// TIA Portal project "Traffic Light Controller" (V16)

(* hardware
DEVICE "S7-1200 station_1"  S7-1200 Station
   slot 0: "Rack_0"  S7-1200 Rack  Rack  V1.0
   slot 1: "PLC_1"  CPU 1212C DC/DC/DC  6ES7 212-1AE40-0XB0  V4.4
DEVICE "HMI_1"  TP700 Comfort
   slot 0: "HMI_1"  TP700 Comfort  6AV2 124-0GC01-0AX0  16.0.0.0
   slot 1: "HMI_RT_1"  TP700 Comfort  6AV2 124-0GC01-0AX0  16.0.0.0
   slot 5: "HMI_1.IE_CP_1"  PROFINET Interface  16.0.0.0
      slot 1: "PROFINET Interface_1"  PROFINET Interface
         slot 1: "Port_1"  Port
         slot 2: "Port_2"  Port
   slot 7: "HMI_1.MPI/DP_CP_1"  MPI/DP Interface  16.0.0.0
*)

// ===== PLC "PLC_1"  CPU 1212C DC/DC/DC =====

VAR_GLOBAL   // PLC tag table "Tag table_1"
   "START" AT %M0.0 : Bool;
   "STOP" AT %M0.1 : Bool;
   "STARTED" AT %M0.2 : Bool;
   "STEP1_EAST_GREEN" AT %M0.3 : Bool;
   "STEP1_WEST_RED" AT %M0.4 : Bool;
   "STEP1_NORTH_RED" AT %M0.5 : Bool;
   "STEP1_EAST_YELLOW" AT %M0.6 : Bool;
   "STEP1_FINISHED" AT %M0.7 : Bool;
   "STEP2_WEST_GREEN" AT %M1.0 : Bool;
   "STEP2_EAST_RED" AT %M1.1 : Bool;
   "STEP2_NORTH_RED" AT %M1.2 : Bool;
   "STEP2_WEST_YELLOW" AT %M1.3 : Bool;
   "STEP2_FINISHED" AT %M1.4 : Bool;
   "STEP3_NORTH_GREEN" AT %M1.5 : Bool;
   "STEP3_EAST_RED" AT %M1.6 : Bool;
   "STEP3_WEST_RED" AT %M1.7 : Bool;
   "STEP3_NORTH_YELLOW" AT %M2.0 : Bool;
   "STEP3_FINISHED" AT %M2.1 : Bool;
   "EAST_GREEN" AT %M2.2 : Bool;
   "EAST_RED" AT %M2.4 : Bool;
   "NORTH_RED" AT %M2.5 : Bool;
   "NORTH_YELLOW" AT %M2.6 : Bool;
   "NORTH_GREEN" AT %M2.7 : Bool;
   "WEST_RED" AT %M3.0 : Bool;
   "WEST_GREEN" AT %M3.1 : Bool;
   "WEST_YELLOW" AT %M3.2 : Bool;
   "EAST_YELLOW" AT %M2.3 : Bool;
END_VAR

// folder: System blocks/Program resources

DATA_BLOCK "STEP1"   // DB1
{ S7_Optimized_Access := 'TRUE' }
AUTHOR : Simatic
FAMILY : IEC
NAME : IEC_TMR
VERSION : 1.0
// stored: InstanceOfName IEC_TIMER
"IEC_TIMER"
BEGIN
END_DATA_BLOCK

DATA_BLOCK "COUNTER_STEP"   // DB2
{ S7_Optimized_Access := 'TRUE' }
AUTHOR : Simatic
FAMILY : IEC
NAME : CNTR
VERSION : 1.0
// stored: InstanceOfName IEC_COUNTER
"IEC_COUNTER"
BEGIN
END_DATA_BLOCK

DATA_BLOCK "STEP2"   // DB3
{ S7_Optimized_Access := 'TRUE' }
AUTHOR : Simatic
FAMILY : IEC
NAME : IEC_TMR
VERSION : 1.0
// stored: InstanceOfName IEC_TIMER
"IEC_TIMER"
BEGIN
END_DATA_BLOCK

DATA_BLOCK "STEP3"   // DB4
{ S7_Optimized_Access := 'TRUE' }
AUTHOR : Simatic
FAMILY : IEC
NAME : IEC_TMR
VERSION : 1.0
// stored: InstanceOfName IEC_TIMER
"IEC_TIMER"
BEGIN
END_DATA_BLOCK

// folder: (top level)

ORGANIZATION_BLOCK "Main"   // OB1, LAD, ProgramCycle
TITLE = "Main Program Sweep (Cycle)"
{ S7_Optimized_Access := 'TRUE' }
VERSION : 0.1
   VAR_INPUT
      Initial_Call : Bool;   // Initial call of this OB
      Remanence : Bool;   // =True, if remanent data are available
   END_VAR
   VAR_TEMP   // added for the SCL form of the ladder/FBD networks
      _w1 : Bool;
      _w2 : Bool;
      _w3 : Bool;
   END_VAR
BEGIN

REGION Network 1
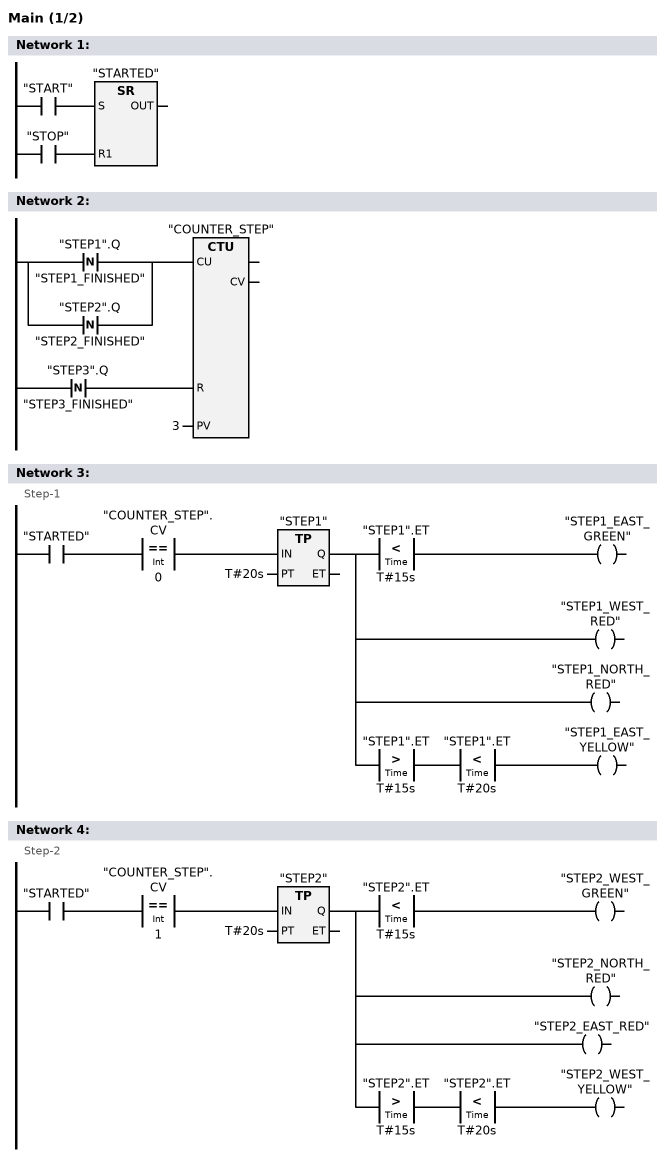
   RUNG wire#powerrail
      Contact( "START" )
      S_SR(operand := "STARTED", r1 := wire#w1)
   END_RUNG
   RUNG wire#powerrail
      Contact( "STOP" )
   END_RUNG wire#w1
   // the same network as SCL:
   IF "START" THEN
       "STARTED" := TRUE;   // SR flip-flop
   END_IF;
   IF "STOP" THEN "STARTED" := FALSE; END_IF;
END_REGION

REGION Network 2
   #_w1 := NOT "STEP1".Q AND "STEP1_FINISHED";   // falling edge of "STEP1".Q
   "STEP1_FINISHED" := "STEP1".Q;
   #_w2 := NOT "STEP2".Q AND "STEP2_FINISHED";   // falling edge of "STEP2".Q
   "STEP2_FINISHED" := "STEP2".Q;
   #_w3 := NOT "STEP3".Q AND "STEP3_FINISHED";   // falling edge of "STEP3".Q
   "STEP3_FINISHED" := "STEP3".Q;
   "COUNTER_STEP".CTU(CU := #_w1 OR #_w2, R := #_w3, PV := 3);
END_REGION

REGION Network 3
   // Step-1
   "STEP1".TP(IN := "STARTED" AND ("COUNTER_STEP".CV = 0), PT := T#20s);
   "STEP1_EAST_GREEN" := "STEP1".Q AND ("STEP1".ET < T#15s);
   "STEP1_WEST_RED" := "STEP1".Q;
   "STEP1_NORTH_RED" := "STEP1".Q;
   "STEP1_EAST_YELLOW" := "STEP1".Q AND ("STEP1".ET > T#15s) AND ("STEP1".ET < T#20s);
END_REGION

REGION Network 4
   // Step-2
   "STEP2".TP(IN := "STARTED" AND ("COUNTER_STEP".CV = 1), PT := T#20s);
   "STEP2_WEST_GREEN" := "STEP2".Q AND ("STEP2".ET < T#15s);
   "STEP2_NORTH_RED" := "STEP2".Q;
   "STEP2_EAST_RED" := "STEP2".Q;
   "STEP2_WEST_YELLOW" := "STEP2".Q AND ("STEP2".ET > T#15s) AND ("STEP2".ET < T#20s);
END_REGION

REGION Network 5
   // Step-3
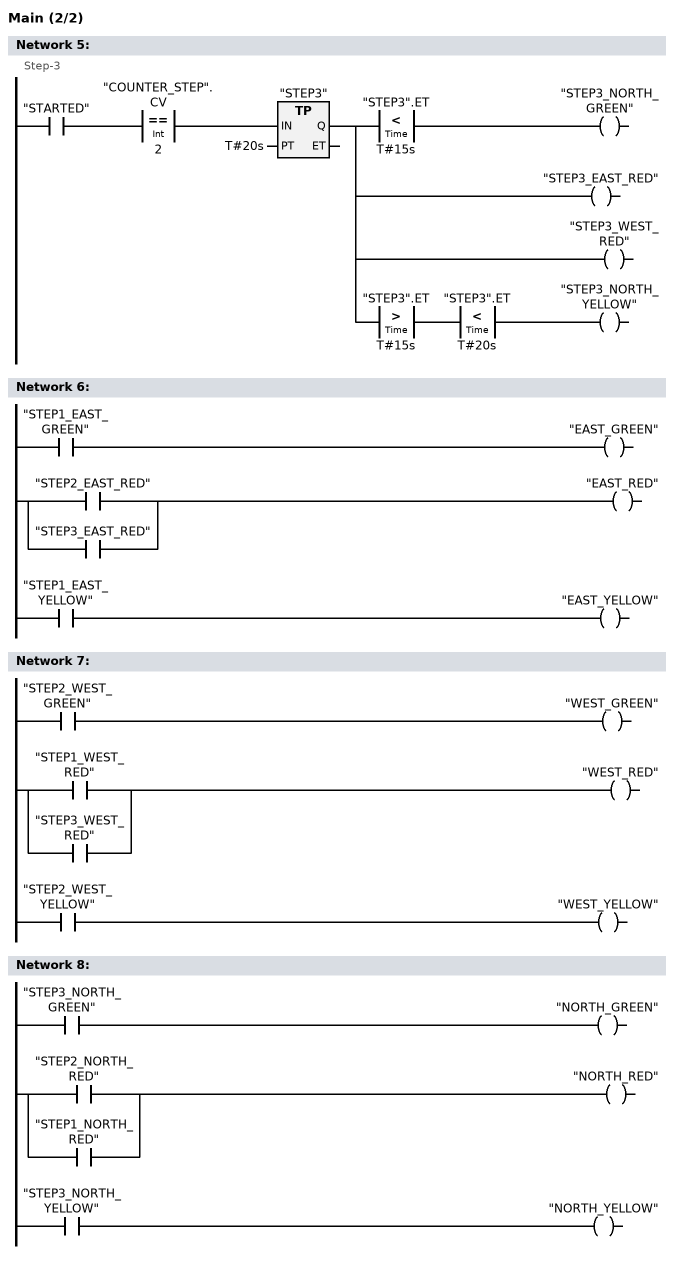
   "STEP3".TP(IN := "STARTED" AND ("COUNTER_STEP".CV = 2), PT := T#20s);
   "STEP3_NORTH_GREEN" := "STEP3".Q AND ("STEP3".ET < T#15s);
   "STEP3_EAST_RED" := "STEP3".Q;
   "STEP3_WEST_RED" := "STEP3".Q;
   "STEP3_NORTH_YELLOW" := "STEP3".Q AND ("STEP3".ET > T#15s) AND ("STEP3".ET < T#20s);
END_REGION

REGION Network 6
   RUNG wire#powerrail
      Contact( "STEP1_EAST_GREEN" )
      Coil( "EAST_GREEN" )
   END_RUNG
   RUNG wire#powerrail
      Contact( "STEP2_EAST_RED" )
      wire#w1
      Coil( "EAST_RED" )
   END_RUNG
   RUNG wire#powerrail
      Contact( "STEP3_EAST_RED" )
   END_RUNG wire#w1
   RUNG wire#powerrail
      Contact( "STEP1_EAST_YELLOW" )
      Coil( "EAST_YELLOW" )
   END_RUNG
   // the same network as SCL:
   "EAST_GREEN" := "STEP1_EAST_GREEN";
   "EAST_RED" := "STEP2_EAST_RED" OR "STEP3_EAST_RED";
   "EAST_YELLOW" := "STEP1_EAST_YELLOW";
END_REGION

REGION Network 7
   RUNG wire#powerrail
      Contact( "STEP2_WEST_GREEN" )
      Coil( "WEST_GREEN" )
   END_RUNG
   RUNG wire#powerrail
      Contact( "STEP1_WEST_RED" )
      wire#w1
      Coil( "WEST_RED" )
   END_RUNG
   RUNG wire#powerrail
      Contact( "STEP3_WEST_RED" )
   END_RUNG wire#w1
   RUNG wire#powerrail
      Contact( "STEP2_WEST_YELLOW" )
      Coil( "WEST_YELLOW" )
   END_RUNG
   // the same network as SCL:
   "WEST_GREEN" := "STEP2_WEST_GREEN";
   "WEST_RED" := "STEP1_WEST_RED" OR "STEP3_WEST_RED";
   "WEST_YELLOW" := "STEP2_WEST_YELLOW";
END_REGION

REGION Network 8
   RUNG wire#powerrail
      Contact( "STEP3_NORTH_GREEN" )
      Coil( "NORTH_GREEN" )
   END_RUNG
   RUNG wire#powerrail
      Contact( "STEP2_NORTH_RED" )
      wire#w1
      Coil( "NORTH_RED" )
   END_RUNG
   RUNG wire#powerrail
      Contact( "STEP1_NORTH_RED" )
   END_RUNG wire#w1
   RUNG wire#powerrail
      Contact( "STEP3_NORTH_YELLOW" )
      Coil( "NORTH_YELLOW" )
   END_RUNG
   // the same network as SCL:
   "NORTH_GREEN" := "STEP3_NORTH_GREEN";
   "NORTH_RED" := "STEP2_NORTH_RED" OR "STEP1_NORTH_RED";
   "NORTH_YELLOW" := "STEP3_NORTH_YELLOW";
END_REGION
END_ORGANIZATION_BLOCK

(* ===== HMI "HMI_RT_1" =====
system functions are stored by id; their names below are inferred from use
connection "HMI_Connection_1": ETHERNET, S7_1200_OMS

HMI tags "Default tag table"
   "WEST_GREEN" : Bool = PLC WEST_GREEN AT %M3.1, 1 s
   "WEST_YELLOW" : Bool = PLC WEST_YELLOW AT %M3.2, 1 s
   "WEST_RED" : Bool = PLC WEST_RED AT %M3.0, 1 s
   "NORTH_GREEN" : Bool = PLC NORTH_GREEN AT %M2.7, 1 s
   "NORTH_YELLOW" : Bool = PLC NORTH_YELLOW AT %M2.6, 1 s
   "NORTH_RED" : Bool = PLC NORTH_RED AT %M2.5, 1 s
   "EAST_YELLOW" : Bool = PLC EAST_YELLOW AT %M2.3, 1 s
   "EAST_RED" : Bool = PLC EAST_RED AT %M2.4, 1 s
   "START" : Bool = PLC START AT %M0.0, 1 s
   "STOP" : Bool = PLC STOP AT %M0.1, 1 s
   "EAST_GREEN" : Bool = PLC EAST_GREEN AT %M2.2, 1 s

screen "Screen_1" 800x480
   Button "Button_1" at 244,46 size 230x44; TextOff 'Text'
   Button "Button_2" at 64,140 size 54x171; TextOff 'Text'
   Button "Button_3" at 612,128 size 60x189; TextOff 'Text'
   TextField "Text field_1" at 79,193 size 28x64; Text 'WEST'
   TextField "Text field_2" at 626,186 size 28x57; Text 'EAST'
   TextField "Text field_3" at 305,52 size 81x27; Text 'NORTH'
   GraphicView "Graphic view_1" at 494,235 size 52x45; Picture "CAR2"
   GraphicView "Graphic view_2" at 168,179 size 47x48; Picture "CAR1"
   GraphicView "Graphic view_3" at 167,234 size 52x45; Picture "CAR2"
   GraphicView "Graphic view_4" at 382,88 size 53x56; Picture "CAR3"
   GraphicView "Graphic view_5" at 302,106 size 53x56; Picture "CAR3"
   Circle "Circle_12" at 391,156 size 16x16
      Appearance <- "NORTH_GREEN"
   Circle "Circle_14" at 408,157 size 16x16
      Appearance <- "NORTH_YELLOW"
   Circle "Circle_15" at 431,157 size 16x16
      Appearance <- "NORTH_RED"
   Circle "Circle_17" at 440,263 size 16x16
      Appearance <- "EAST_RED"
   Circle "Circle_18" at 440,247 size 16x16
      Appearance <- "EAST_YELLOW"
   Circle "Circle_19" at 440,231 size 16x16
      Appearance <- "EAST_GREEN"
   Circle "Circle_20" at 274,178 size 16x16
      Appearance <- "WEST_GREEN"
   Circle "Circle_21" at 274,196 size 16x16
      Appearance <- "WEST_YELLOW"
   Circle "Circle_22" at 274,213 size 16x16
      Appearance <- "WEST_RED"
   Button "Button_4" at 672,9 size 96x32; TextOff 'START'
      on Press: SetBit("START")
      on Release: ResetBit("START")
   Button "Button_5" at 672,52 size 96x32; TextOff 'STOP'
      on Press: SetBit("STOP")
      on Release: ResetBit("STOP")
*)